{attribute 'GeneratedUsingTerminal: EPP1321-0060-0016'}
{attribute addProperty BoxType "EPP1321-0060-0016"}
{attribute addProperty Id "A_0019_EPP1322_0001_0016A_0019_EPP1322_0001_0016_AC0682C2378"}
{attribute addProperty CRC "3084128359"}
{attribute addProperty Size "378"}
TYPE A_0018_EPP1321_0060_0016_B7D41067 EXTENDS EPP1321_AB5A9467 :
STRUCT
	{attribute addProperty Name "A_0019_EPP1322_0001_0016"}
	{attribute addProperty PreviousPort "A_0018(EPP1321-0060-0016) : D"}
	A_0019_EPP1322_0001_0016 : A_0019_EPP1322_0001_0016_AC0682C2;
END_STRUCT
END_TYPE

(* stored: Version 1.2.0.0, ProductVersion 3.1.4024.9
   DUT A_0018_EPP1321_0060_0016_B7D41067: Id {82be2632-b1bf-4127-98a9-9a496d19a9c5} *)
